TYPE ST_Chamber1_ServiceStatus :
STRUCT
	SpinAxisJogCW : ST_ServiceStatus;
	SpinAxisMoveAbs : ST_ServiceStatus;
	SpinAxisMoveVelCW : ST_ServiceStatus;
	LiftPinAxisMoveVelCW : ST_ServiceStatus;
	LiftPinAxisMoveVelCCW : ST_ServiceStatus;
	LiftPinAxisMoveAbs : ST_ServiceStatus;
	SingleProcess : ST_ServiceStatus;
	WaferSend : ST_ServiceStatus;
	WaferReceive : ST_ServiceStatus;
	PreparePosition : ST_ServiceStatus;
END_STRUCT
END_TYPE

(* stored: Version 1.1.0.1, ProductVersion 3.1.4026.18
   DUT ST_Chamber1_ServiceStatus: Id {f27be8ff-16cd-4df7-a4df-6e0527b043a3} *)
